{attribute 'GeneratedUsingTerminal: EL3751-0000-0020'}
{attribute addProperty BoxType "EL3751-0000-0020"}
{attribute addProperty Id "No_of_SamplesUSINT1ErrorBOOL1UnderrangeBOOL1OverrangeBOOL1DiagBOOL1TxPDO_StateBOOL1Input_cycle_counterBYTE1"}
{attribute addProperty CRC "1412436158"}
{attribute addProperty Size "7"}
TYPE Status_543010BE :
STRUCT
	{attribute addProperty Name "No_of_Samples"}
	No_of_Samples : USINT;
	{attribute addProperty Name "Error"}
	Error : BOOL;
	{attribute addProperty Name "Underrange"}
	Underrange : BOOL;
	{attribute addProperty Name "Overrange"}
	Overrange : BOOL;
	{attribute addProperty Name "Diag"}
	Diag : BOOL;
	{attribute addProperty Name "TxPDO_State"}
	TxPDO_State : BOOL;
	{attribute addProperty Name "Input_cycle_counter"}
	Input_cycle_counter : BYTE;
END_STRUCT
END_TYPE

(* stored: Version 1.2.0.0, ProductVersion 3.1.4024.11
   DUT Status_543010BE: Id {98b8ed71-468e-4ec1-82fa-ff444b76f6d5} *)
